TEXTLIST CtrlModeTextList
  1 = '自动模式' | Chinese: '自动模式' | English: 'Auto Mode'
  2 = '手动模式' | Chinese: '手动模式' | English: 'Manual Mode'
  3 = '调试模式' | Chinese: '调试模式' | English: 'Debug Mode'
  9 = '配置模式' | Chinese: '配置模式' | English: 'Config Mode'
   = ''
END_TEXTLIST

(* stored: Version 1.1.0.1, ProductVersion 3.1.4024.4
   TextList CtrlModeTextList: Id {e4f8be30-58f9-44e9-ba04-54a46d8e6e6b} *)
